PROGRAM GVL
VAR
END_VAR

END_PROGRAM

(* stored: Version 1.1.0.1, ProductVersion 3.1.4024.10
   POU GVL: Id {eac86cfe-cb67-4d23-9bd9-0c199b371614}, SpecialFunc None *)
